PROGRAM MAIN
VAR
END_VAR

END_PROGRAM

(* stored: Version 1.1.0.1
   POU MAIN: Id {982bde0f-179e-4b17-b613-c9f5863bc8c6} *)
